(* Logix 5000 project; controller Safety vendor 1 type 14 code 86 rev 19.11; software revision 19.01; part 5 of 17 *)
(* tags used below, declared in another part *)
   A1_CoilCarSolPwrEn : BOOL;   // A1 UNW COIL CAR Solenoid Safe-Off Enable ( 1= Enable )
   ChgMe : BOOL;
   DAM : ALIAS FOR Diag_Tmp.4;   // Doug M Always Off Test Bit
   FltsToCitect : DINT[64];   // Faults to Citect
   FromCitect : DINT[64];   // (From Citect)
   FromMach : DINT[35];   // (FromMach)
   FromMachine : DINT[35];   // (FromMach)
   FromSafety : DINT[35];   // (From Safety)
   FromShearDie : DINT[35];   // (From Shear Die)
   FUTURE : ALIAS FOR Diag_Tmp.1;   // FUTURE
   LineSts : UDT_SysStatus;
   Map_Citect : DINT[5];   // Mapped From Shear Citect System
   Map_Mach : DINT[5];   // From Machine Processor
   Map_ShDie : DINT[5];   // Mapped From Shear Die Processor
   SafeOff_y172CR510 : CONFIGURABLE_ROUT;   // Shear Die Drive Enable Relay
   SafeOff_y613CR510 : CONFIGURABLE_ROUT;   // Unwind Op Side Drive Enable Relay
   SafeOff_y613CR550 : CONFIGURABLE_ROUT;   // Unwind Drive Side Main Contactor Relay
   SafeOff_y613CR670 : CONFIGURABLE_ROUT;   // #1 Entry Bridle Roll 2 Drive Enable Relay
   SafeOff_y613CR750 : CONFIGURABLE_ROUT;   // #2 Entry Bridle Roll 3 Drive Enable Relay
   SafeOff_y614CR090 : CONFIGURABLE_ROUT;   // #1 Exit Bridle Roll 6 Drive Enable Relay
   SafeOff_y614CR170 : CONFIGURABLE_ROUT;   // #2 Exit Bridle Roll 7 Drive Enable Relay
   SafeOff_y614CR250 : CONFIGURABLE_ROUT;   // Rewind Drive Enable Relay
   SftyMap_Citect : DINT[5];   // SAFETY MAPPED From Citect System
   SftyMap_Mach : DINT[5];   // SAFETY MAPPED From Machine Processor
   SftyMap_ShDie : DINT[5];   // SAFETY MAPPED From Shear Die Processor
   ShearSts : UDT_ShearStatus;
   ToCitect : DINT[64];   // (To Citect)
   ToCitect4 : DINT[64];   // (To Citect4)
   x702MTR191FF : ALIAS FOR MCC1:1:I.Pt00Data;   // Rewind Pinch Roll Fwd Fdbk
   x702MTR191RF : ALIAS FOR MCC1:1:I.Pt01Data;   // Rewind Pinch Roll Rev Fdbk
   x708MTR080FF : ALIAS FOR MCC1:1:I.Pt04Data;   // Flattener Drive Motor Fwd Fdbk
   x708MTR080RF : ALIAS FOR MCC1:1:I.Pt05Data;   // Flattener Drive Motor Rev Fdbk
   x708MTR250FF : ALIAS FOR MCC1:1:I.Pt06Data;   // Unwind Holddown Roll Drive Motor Fwd Fdbk
   x708MTR250RF : ALIAS FOR MCC1:1:I.Pt07Data;   // Unwind Holddown Roll Drive Motor Rev Fdbk
   x753MTR190FF : ALIAS FOR MCC3:1:I.Pt00Data;   // Trimmer Pinch Roll Fwd Fdbk
   x753MTR190RF : ALIAS FOR MCC3:1:I.Pt01Data;   // Trimmer Pinch Roll Rev Fdbk
   x759MTR080SE : ALIAS FOR MCC3:4:O.Pt02Data;   // Scrap Choppers Width Adjust Safety Enable
   x761MTR081RF : ALIAS FOR MCC3:1:I.Pt02Data;   // Trimmer Scrap Conveyor RunFdbk
   x778MTR080RF : ALIAS FOR MCC4:1:I.Pt00Data;   // Shear Crank Motor Run Fdbk
   x802MTR080FF : ALIAS FOR MCC5:1:I.Pt00Data;   // Stacker Side Guide Lift Fwd Fdbk/Up
   x802MTR080RF : ALIAS FOR MCC5:1:I.Pt01Data;   // Stacker Side Guide Lift Rev Fdbk/Down
   x802MTR230FF : ALIAS FOR MCC5:1:I.Pt02Data;   // Scrap Horizontal Conveyor Run Fwd Fdbk
   x802MTR230RF : ALIAS FOR MCC5:1:I.Pt03Data;   // Scrap Horizontal Conveyor Run Rev Fdbk
   x802MTR231FF : ALIAS FOR MCC5:1:I.Pt04Data;   // Stacker Chain Fwd Fdbk
   x802MTR231RF : ALIAS FOR MCC5:1:I.Pt05Data;   // Stacker Chain Rev Fdbk
   y725MTR080SE : ALIAS FOR MCC2:1:O.Pt01Data;   // Unwind Pinch Roll Safety Enable
   y727MTR080SE : ALIAS FOR MCC2:1:O.Pt05Data;   // Paper Winder Safety Enable
   y729MTR080SE : ALIAS FOR MCC2:1:O.Pt03Data;   // Washtank Pinch Roll 4 Safety Enable
   y731MTR080SE : ALIAS FOR MCC2:1:O.Pt07Data;   // Washtank Pinch Roll 1 Safety Enable
   y733MTR080SE : ALIAS FOR MCC2:2:O.Pt01Data;   // Washtank Pinch Roll 2 Safety Enable
   y735MTR080SE : ALIAS FOR MCC2:2:O.Pt03Data;   // Washtank Pinch Roll 3 Safety Enable
   y751MTR080SE : ALIAS FOR MCC3:3:O.Pt04Data;   // Trimmer Knives Safety Enable
   y754MTR080SE : ALIAS FOR MCC3:3:O.Pt06Data;   // Side Guide Width Adjust Safety Enable
   y755MTR080SE : ALIAS FOR MCC3:4:O.Pt00Data;   // Trimmer Knives Width Adjust Safety Enable
   y762MTR080SE : ALIAS FOR MCC3:4:O.Pt04Data;   // Scrap Choppers Safety Enable
   y776MTR080SE : ALIAS FOR MCC4:3:O.Pt07Data;   // Shear Metering Backup Roll Safety Enable
   y779MTR080SE : ALIAS FOR MCC4:3:O.Pt01Data;   // Shear Pinch Roll Safety Enable
   y782MTR080SE : ALIAS FOR MCC4:3:O.Pt03Data;   // Sheeter Pinch Roll Safety Enable
   y785MTR080SE : ALIAS FOR MCC4:3:O.Pt05Data;   // Stacker Blower Safety Enable
   y800MTR080SE : ALIAS FOR MCC5:3:O.Pt01Data;   // Scrap Incline Conveyor Safety Enable
   y804MTR080SE : ALIAS FOR MCC5:3:O.Pt03Data;   // Stacker Back Stop Safety Enable
   y806MTR080SE : ALIAS FOR MCC5:3:O.Pt05Data;   // Product Conveyor 3 Safety Enable
   y808MTR080SE : ALIAS FOR MCC5:3:O.Pt07Data;   // Product Conveyor 1 Safety Enable
   y810MTR080SE : ALIAS FOR MCC5:4:O.Pt01Data;   // Product Conveyor 2 Safety Enable
   y812MTR080SE : ALIAS FOR MCC5:4:O.Pt03Data;   // Shear Conveyor Safety Enable
(* Comms, continued *)

ROUTINE MainRoutine   (* ladder *)
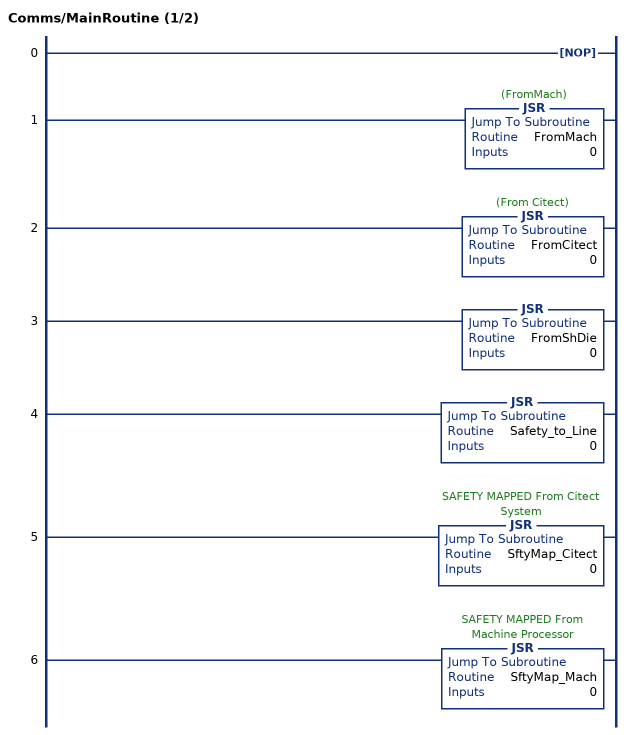
   0: NOP();
   1: JSR(FromMach,0);
   2: JSR(FromCitect,0);
   3: JSR(FromShDie,0);
   4: JSR(Safety_to_Line,0);
   5: JSR(SftyMap_Citect,0);
   6: JSR(SftyMap_Mach,0);
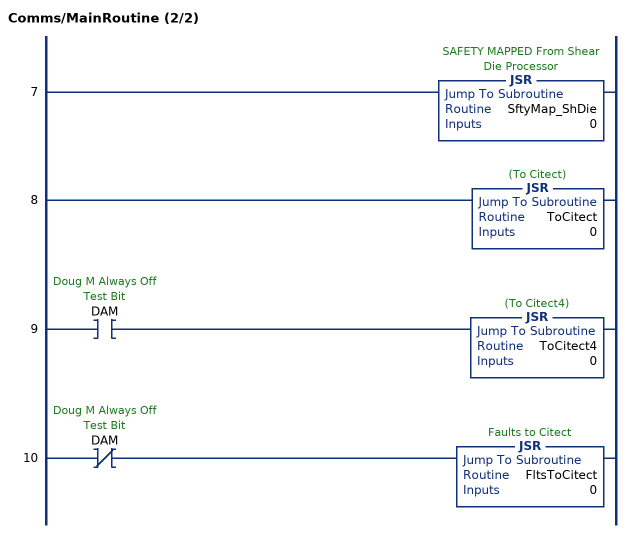
   7: JSR(SftyMap_ShDie,0);
   8: JSR(ToCitect,0);
   9: XIC(DAM)JSR(ToCitect4,0);
   10: XIO(DAM)JSR(FltsToCitect,0);
END_ROUTINE

ROUTINE Safety_to_Line   (* ladder *)
// Safety Signals to Line
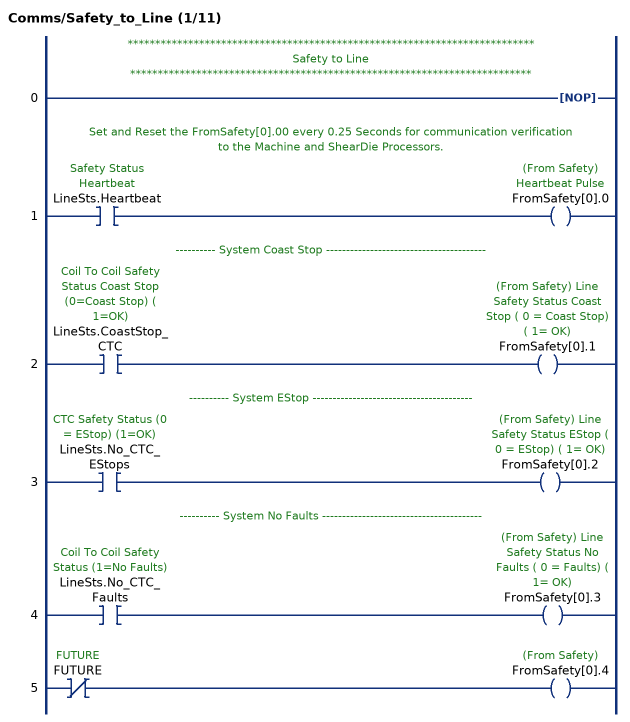
   // **************************************************************************
   // Safety to Line
   // *************************************************************************
   0: NOP();
   // Set and Reset the FromSafety[0].00 every 0.25 Seconds for communication verification
   // to the Machine and ShearDie Processors.
   1: XIC(LineSts.Heartbeat)OTE(FromSafety[0].0);
   // ---------- System Coast Stop ----------------------------------------
   2: XIC(LineSts.CoastStop_CTC)OTE(FromSafety[0].1);
   // ---------- System EStop ----------------------------------------
   3: XIC(LineSts.No_CTC_EStops)OTE(FromSafety[0].2);
   // ---------- System No Faults ----------------------------------------
   4: XIC(LineSts.No_CTC_Faults)OTE(FromSafety[0].3);
   5: XIO(FUTURE)OTE(FromSafety[0].4);
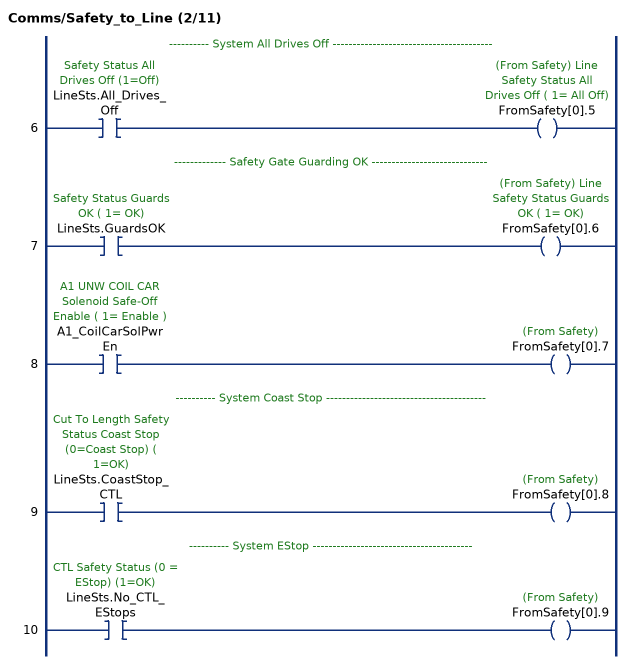
   // ---------- System All Drives Off ----------------------------------------
   6: XIC(LineSts.All_Drives_Off)OTE(FromSafety[0].5);
   // ------------- Safety Gate Guarding OK -----------------------------
   7: XIC(LineSts.GuardsOK)OTE(FromSafety[0].6);
   8: XIC(A1_CoilCarSolPwrEn)OTE(FromSafety[0].7);
   // ---------- System Coast Stop ----------------------------------------
   9: XIC(LineSts.CoastStop_CTL)OTE(FromSafety[0].8);
   // ---------- System EStop ----------------------------------------
   10: XIC(LineSts.No_CTL_EStops)OTE(FromSafety[0].9);
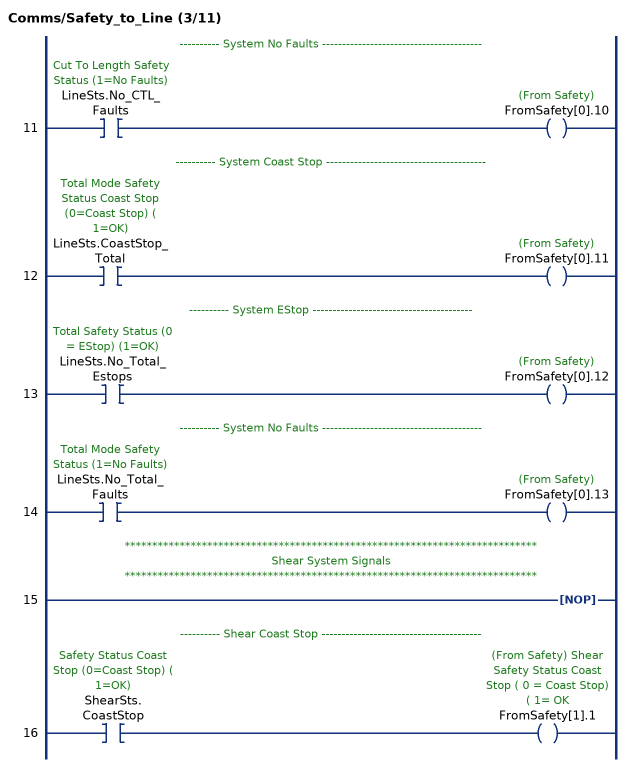
   // ---------- System No Faults ----------------------------------------
   11: XIC(LineSts.No_CTL_Faults)OTE(FromSafety[0].10);
   // ---------- System Coast Stop ----------------------------------------
   12: XIC(LineSts.CoastStop_Total)OTE(FromSafety[0].11);
   // ---------- System EStop ----------------------------------------
   13: XIC(LineSts.No_Total_Estops)OTE(FromSafety[0].12);
   // ---------- System No Faults ----------------------------------------
   14: XIC(LineSts.No_Total_Faults)OTE(FromSafety[0].13);
   // ***************************************************************************
   // Shear System Signals
   // ***************************************************************************
   15: NOP();
   // ---------- Shear Coast Stop ----------------------------------------
   16: XIC(ShearSts.CoastStop)OTE(FromSafety[1].1);
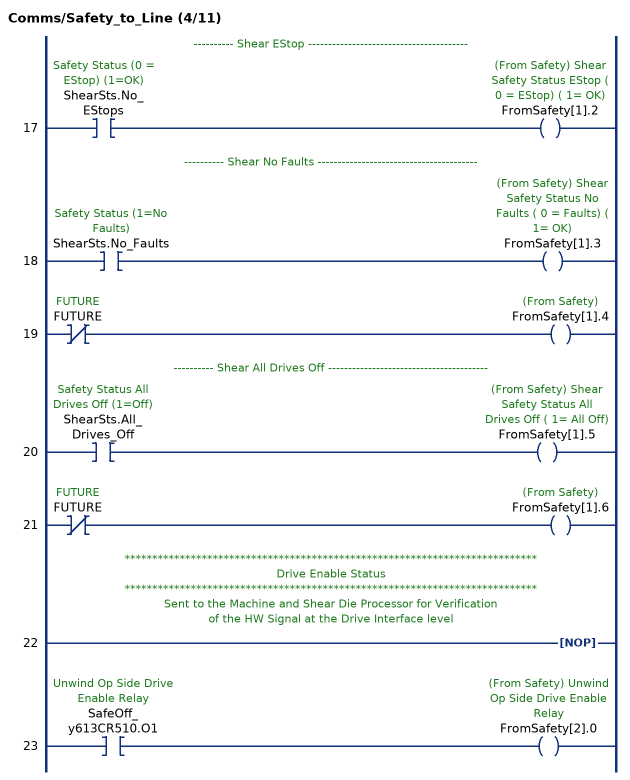
   // ---------- Shear EStop ----------------------------------------
   17: XIC(ShearSts.No_EStops)OTE(FromSafety[1].2);
   // ---------- Shear No Faults ----------------------------------------
   18: XIC(ShearSts.No_Faults)OTE(FromSafety[1].3);
   19: XIO(FUTURE)OTE(FromSafety[1].4);
   // ---------- Shear All Drives Off ----------------------------------------
   20: XIC(ShearSts.All_Drives_Off)OTE(FromSafety[1].5);
   21: XIO(FUTURE)OTE(FromSafety[1].6);
   // ***************************************************************************
   // Drive Enable Status
   // ***************************************************************************
   // Sent to the Machine and Shear Die Processor for Verification
   // of the HW Signal at the Drive Interface level
   22: NOP();
   23: XIC(SafeOff_y613CR510.O1)OTE(FromSafety[2].0);
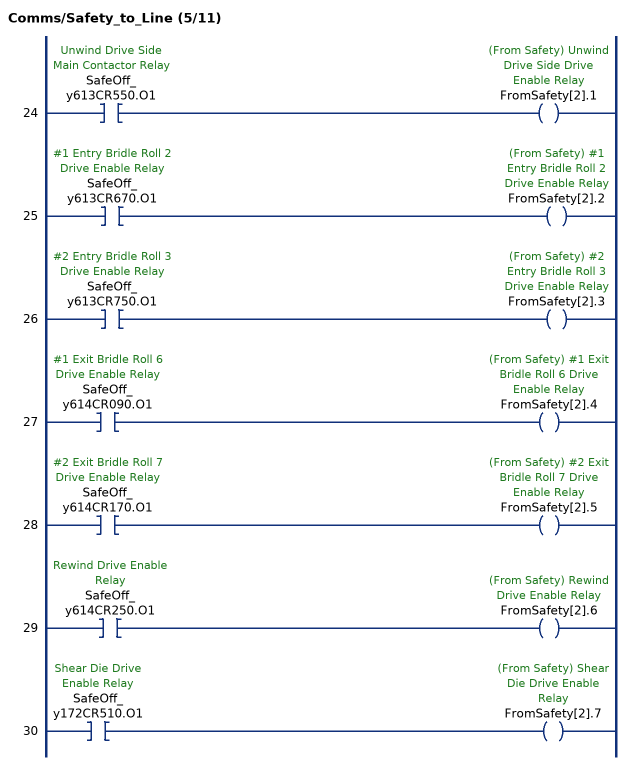
   24: XIC(SafeOff_y613CR550.O1)OTE(FromSafety[2].1);
   25: XIC(SafeOff_y613CR670.O1)OTE(FromSafety[2].2);
   26: XIC(SafeOff_y613CR750.O1)OTE(FromSafety[2].3);
   27: XIC(SafeOff_y614CR090.O1)OTE(FromSafety[2].4);
   28: XIC(SafeOff_y614CR170.O1)OTE(FromSafety[2].5);
   29: XIC(SafeOff_y614CR250.O1)OTE(FromSafety[2].6);
   30: XIC(SafeOff_y172CR510.O1)OTE(FromSafety[2].7);
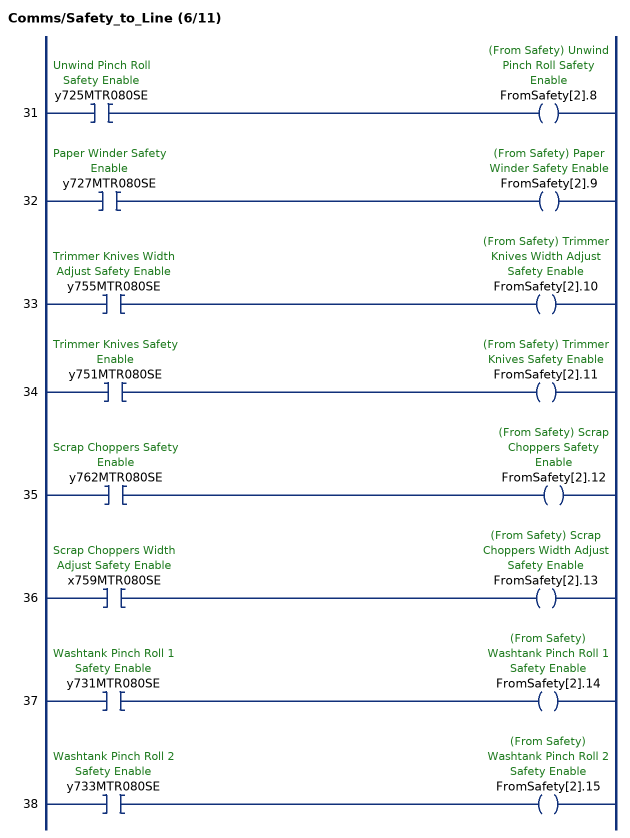
   31: XIC(y725MTR080SE)OTE(FromSafety[2].8);
   32: XIC(y727MTR080SE)OTE(FromSafety[2].9);
   33: XIC(y755MTR080SE)OTE(FromSafety[2].10);
   34: XIC(y751MTR080SE)OTE(FromSafety[2].11);
   35: XIC(y762MTR080SE)OTE(FromSafety[2].12);
   36: XIC(x759MTR080SE)OTE(FromSafety[2].13);
   37: XIC(y731MTR080SE)OTE(FromSafety[2].14);
   38: XIC(y733MTR080SE)OTE(FromSafety[2].15);
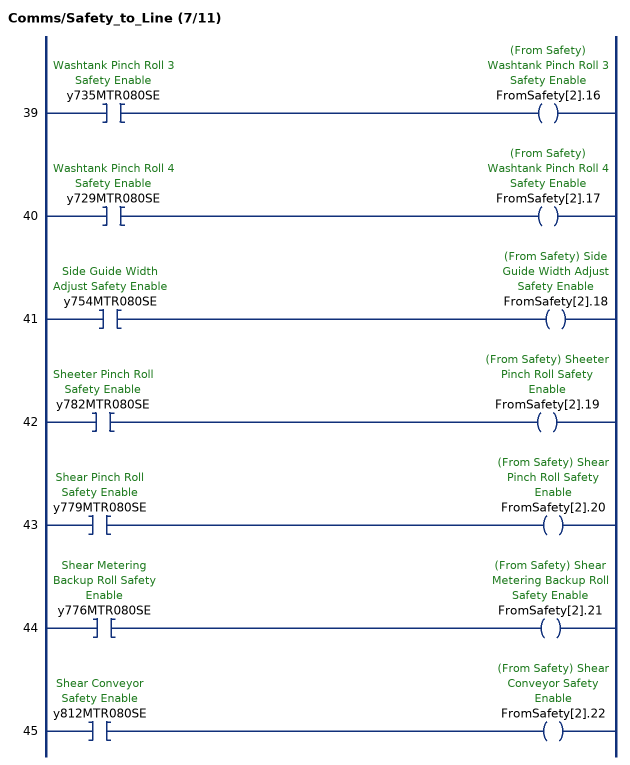
   39: XIC(y735MTR080SE)OTE(FromSafety[2].16);
   40: XIC(y729MTR080SE)OTE(FromSafety[2].17);
   41: XIC(y754MTR080SE)OTE(FromSafety[2].18);
   42: XIC(y782MTR080SE)OTE(FromSafety[2].19);
   43: XIC(y779MTR080SE)OTE(FromSafety[2].20);
   44: XIC(y776MTR080SE)OTE(FromSafety[2].21);
   45: XIC(y812MTR080SE)OTE(FromSafety[2].22);
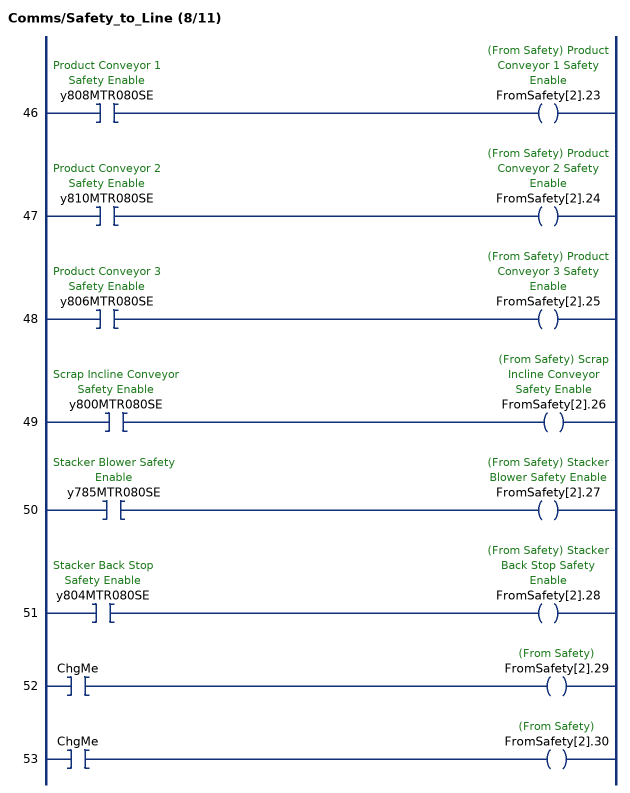
   46: XIC(y808MTR080SE)OTE(FromSafety[2].23);
   47: XIC(y810MTR080SE)OTE(FromSafety[2].24);
   48: XIC(y806MTR080SE)OTE(FromSafety[2].25);
   49: XIC(y800MTR080SE)OTE(FromSafety[2].26);
   50: XIC(y785MTR080SE)OTE(FromSafety[2].27);
   51: XIC(y804MTR080SE)OTE(FromSafety[2].28);
   52: XIC(ChgMe)OTE(FromSafety[2].29);
   53: XIC(ChgMe)OTE(FromSafety[2].30);
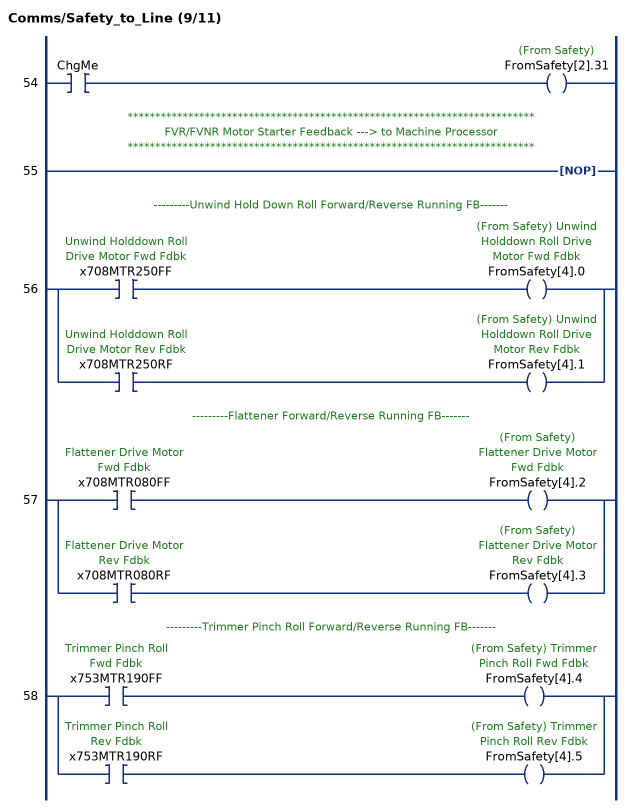
   54: XIC(ChgMe)OTE(FromSafety[2].31);
   // **************************************************************************
   // FVR/FVNR Motor Starter Feedback ---> to Machine Processor
   // **************************************************************************
   55: NOP();
   // ---------Unwind Hold Down Roll Forward/Reverse Running FB-------
   56: [XIC(x708MTR250FF) OTE(FromSafety[4].0) ,XIC(x708MTR250RF) OTE(FromSafety[4].1) ];
   // ---------Flattener Forward/Reverse Running FB-------
   57: [XIC(x708MTR080FF) OTE(FromSafety[4].2) ,XIC(x708MTR080RF) OTE(FromSafety[4].3) ];
   // ---------Trimmer Pinch Roll Forward/Reverse Running FB-------
   58: [XIC(x753MTR190FF) OTE(FromSafety[4].4) ,XIC(x753MTR190RF) OTE(FromSafety[4].5) ];
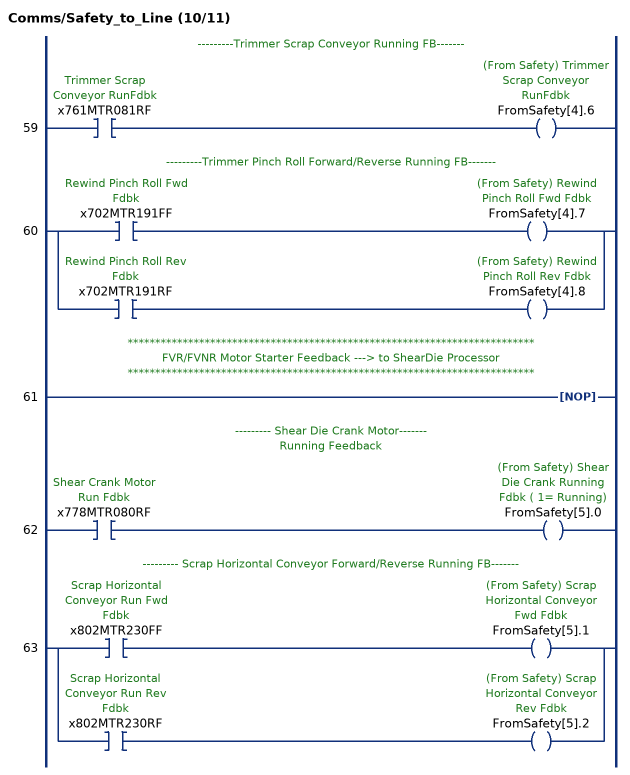
   // ---------Trimmer Scrap Conveyor Running FB-------
   59: XIC(x761MTR081RF)OTE(FromSafety[4].6);
   // ---------Trimmer Pinch Roll Forward/Reverse Running FB-------
   60: [XIC(x702MTR191FF) OTE(FromSafety[4].7) ,XIC(x702MTR191RF) OTE(FromSafety[4].8) ];
   // **************************************************************************
   // FVR/FVNR Motor Starter Feedback ---> to ShearDie Processor
   // **************************************************************************
   61: NOP();
   // --------- Shear Die Crank Motor-------
   // Running Feedback
   62: XIC(x778MTR080RF)OTE(FromSafety[5].0);
   // --------- Scrap Horizontal Conveyor Forward/Reverse Running FB-------
   63: [XIC(x802MTR230FF) OTE(FromSafety[5].1) ,XIC(x802MTR230RF) OTE(FromSafety[5].2) ];
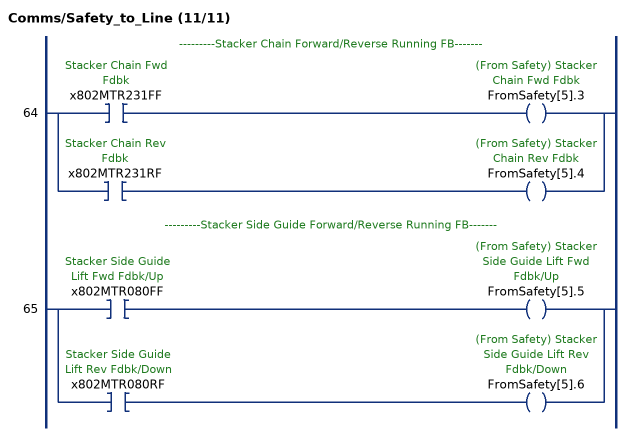
   // ---------Stacker Chain Forward/Reverse Running FB-------
   64: [XIC(x802MTR231FF) OTE(FromSafety[5].3) ,XIC(x802MTR231RF) OTE(FromSafety[5].4) ];
   // ---------Stacker Side Guide Forward/Reverse Running FB-------
   65: [XIC(x802MTR080FF) OTE(FromSafety[5].5) ,XIC(x802MTR080RF) OTE(FromSafety[5].6) ];
END_ROUTINE

ROUTINE SftyMap_Citect   (* ladder *)
// Citect
// Safety Mapped Data
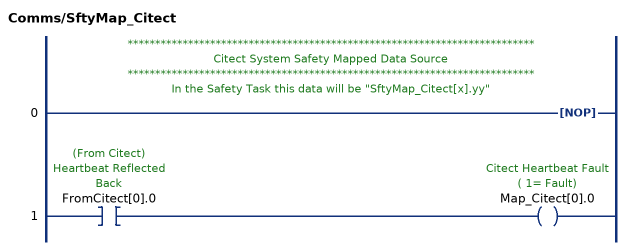
   // **************************************************************************
   // Citect System Safety Mapped Data Source
   // **************************************************************************
   // In the Safety Task this data will be "SftyMap_Citect[x].yy"
   0: NOP();
   1: XIC(FromCitect[0].0)OTE(Map_Citect[0].0);
END_ROUTINE

ROUTINE SftyMap_Mach   (* ladder *)
// Machine
// Safety Mapped Data
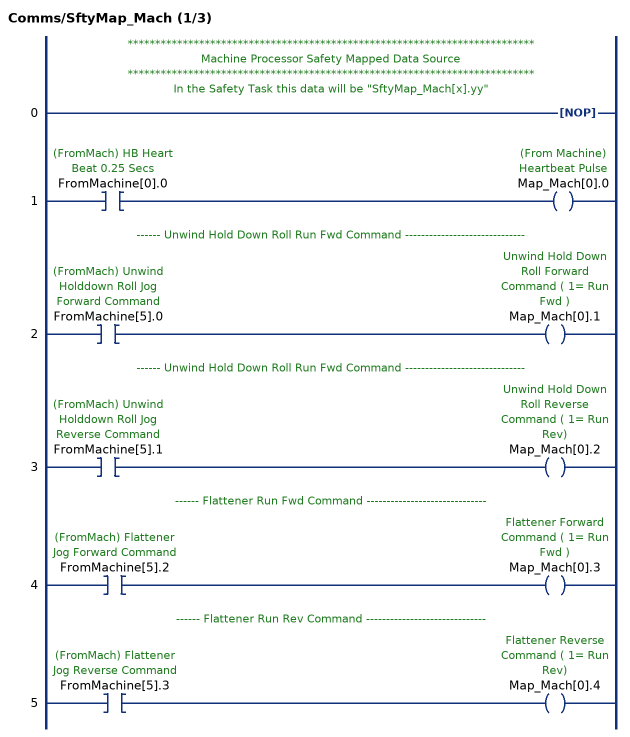
   // **************************************************************************
   // Machine Processor Safety Mapped Data Source
   // **************************************************************************
   // In the Safety Task this data will be "SftyMap_Mach[x].yy"
   0: NOP();
   1: XIC(FromMachine[0].0)OTE(Map_Mach[0].0);
   // ------ Unwind Hold Down Roll Run Fwd Command ------------------------------
   2: XIC(FromMachine[5].0)OTE(Map_Mach[0].1);
   // ------ Unwind Hold Down Roll Run Fwd Command ------------------------------
   3: XIC(FromMachine[5].1)OTE(Map_Mach[0].2);
   // ------ Flattener Run Fwd Command ------------------------------
   4: XIC(FromMachine[5].2)OTE(Map_Mach[0].3);
   // ------ Flattener Run Rev Command ------------------------------
   5: XIC(FromMachine[5].3)OTE(Map_Mach[0].4);
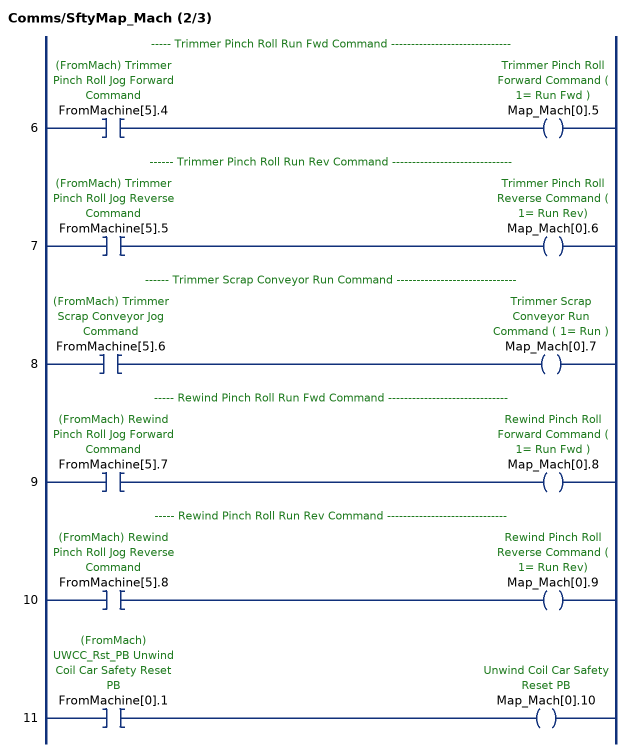
   // ----- Trimmer Pinch Roll Run Fwd Command ------------------------------
   6: XIC(FromMachine[5].4)OTE(Map_Mach[0].5);
   // ------ Trimmer Pinch Roll Run Rev Command ------------------------------
   7: XIC(FromMachine[5].5)OTE(Map_Mach[0].6);
   // ------ Trimmer Scrap Conveyor Run Command ------------------------------
   8: XIC(FromMachine[5].6)OTE(Map_Mach[0].7);
   // ----- Rewind Pinch Roll Run Fwd Command ------------------------------
   9: XIC(FromMachine[5].7)OTE(Map_Mach[0].8);
   // ----- Rewind Pinch Roll Run Rev Command ------------------------------
   10: XIC(FromMachine[5].8)OTE(Map_Mach[0].9);
   11: XIC(FromMachine[0].1)OTE(Map_Mach[0].10);
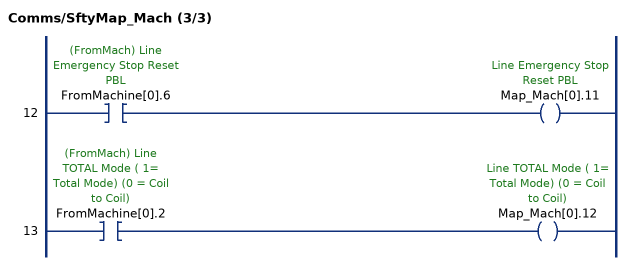
   12: XIC(FromMachine[0].6)OTE(Map_Mach[0].11);
   13: XIC(FromMachine[0].2)OTE(Map_Mach[0].12);
END_ROUTINE

ROUTINE SftyMap_ShDie   (* ladder *)
// Shear Die
// Safety Mapped Data
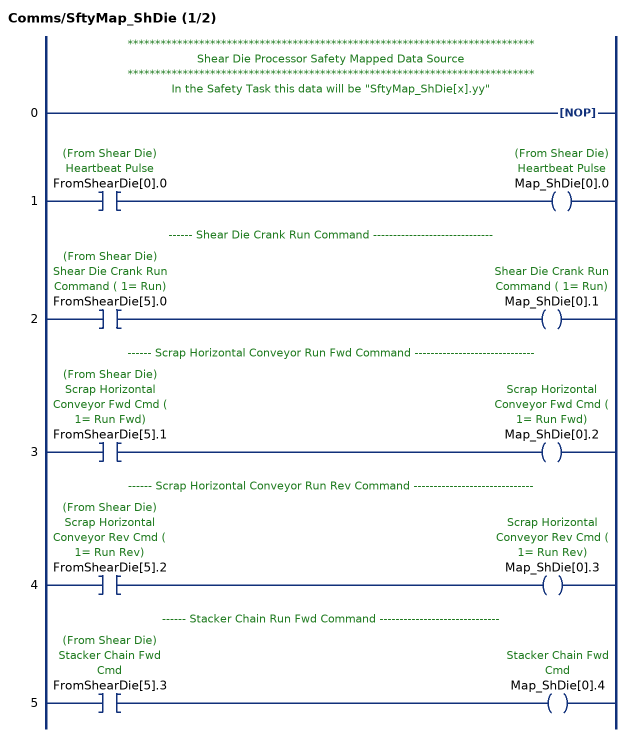
   // **************************************************************************
   // Shear Die Processor Safety Mapped Data Source
   // **************************************************************************
   // In the Safety Task this data will be "SftyMap_ShDie[x].yy"
   0: NOP();
   1: XIC(FromShearDie[0].0)OTE(Map_ShDie[0].0);
   // ------ Shear Die Crank Run Command ------------------------------
   2: XIC(FromShearDie[5].0)OTE(Map_ShDie[0].1);
   // ------ Scrap Horizontal Conveyor Run Fwd Command ------------------------------
   3: XIC(FromShearDie[5].1)OTE(Map_ShDie[0].2);
   // ------ Scrap Horizontal Conveyor Run Rev Command ------------------------------
   4: XIC(FromShearDie[5].2)OTE(Map_ShDie[0].3);
   // ------ Stacker Chain Run Fwd Command ------------------------------
   5: XIC(FromShearDie[5].3)OTE(Map_ShDie[0].4);
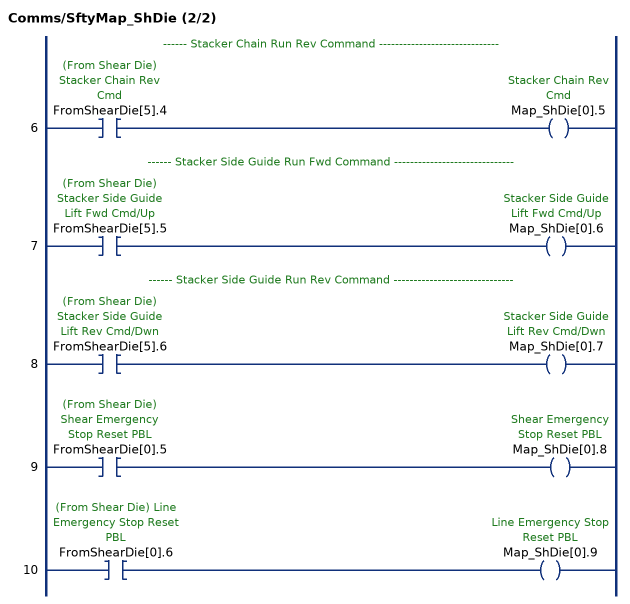
   // ------ Stacker Chain Run Rev Command ------------------------------
   6: XIC(FromShearDie[5].4)OTE(Map_ShDie[0].5);
   // ------ Stacker Side Guide Run Fwd Command ------------------------------
   7: XIC(FromShearDie[5].5)OTE(Map_ShDie[0].6);
   // ------ Stacker Side Guide Run Rev Command ------------------------------
   8: XIC(FromShearDie[5].6)OTE(Map_ShDie[0].7);
   9: XIC(FromShearDie[0].5)OTE(Map_ShDie[0].8);
   10: XIC(FromShearDie[0].6)OTE(Map_ShDie[0].9);
END_ROUTINE
